KUKA KRL data list: ResetaPallet.dat

&ACCESS RVO
&REL 3
&PARAM EDITMASK = *
DEFDAT  ResetaPallet

ENDDAT
